INTERFACE I_InputPortVisitor

METHOD VisitInputPort
VAR_INPUT
	VisitingInputPort : I_InputPort;
END_VAR
END_METHOD

END_INTERFACE

(* stored: Version 1.1.0.1, ProductVersion 3.1.4024.12
   Itf I_InputPortVisitor: Id {cab25b1c-615b-0bc6-1a16-55ee17c0ec1b}
   Method VisitInputPort: Id {6241dbc0-5363-06eb-0faf-c8faa922a437} *)
